Omron CX-Programmer project NewProject (CX-Programmer 9.64)

# PLC CXLiteTestLLB: CJ2H CPU67-EIP
I/O table (CPU CJ2H-CPU67-EIP): rack 0 slot 11 CJ2B-EIP21

## Program NewProgram1 (cyclic task 0)

### Section Section1

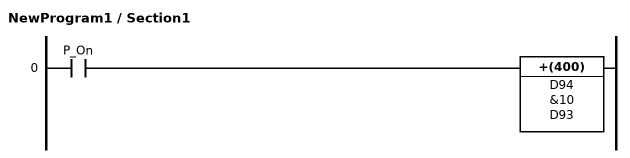
; rung 0
LD P_On
+(400) D94 &10 D93

### Section END
; rung 0
END(001)